// TIA Portal V16 export
// export: Created 2021-11-12T13:32:43.7602296Z, ExportSetting WithDefaults, DisplayName Totally Integrated Automation Portal, DisplayVersion V16 Update 3, DisplayName TIA Portal Version Control Interface, DisplayVersion V16 Update 2, DisplayName TIA Portal Openness, DisplayVersion V16 Update 3, DisplayName SINAMICS Startdrive Advanced, DisplayVersion V16 Update 5, DisplayName SINAMICS Startdrive G130, G150, S120, S150, SINAMICS MV, S210, DisplayVersion V16 Update 5, DisplayName SINAMICS Startdrive G110M, G120, G120C, G120D, G120P, G115D, DisplayVersion V16 Update 5, DisplayName STEP 7 Professional, DisplayVersion V16 Update 3, DisplayName STEP 7 Safety, DisplayVersion V16, DisplayName WinCC UA Professional, DisplayVersion V16 Update 3
DATA_BLOCK "STATUS_SCH1"   // DB51
{ S7_Optimized_Access := 'TRUE' }
VERSION : 0.1
// stored: AutoNumber true, DBAccessibleFromOPCUA true, IsOnlyStoredInLoadMemory false, IsRetainMemResEnabled false, IsWriteProtectedInAS false, MemoryReserve 100
   VAR
      xxxxx___BinarySensors___xxxxx : Byte;
      xxxxx___BinaryOthers___xxxxx : Byte;
      "000UH11-SF05_22" : Bool;   // Blokování lisu
      "000UH10-SF12_22" : Bool;   // Blokování lisu
      "TT1EB01-KF02_4" : Bool;   // Ohřev nástrojů 1 Kontrola chodu čerpadla
      "TT2EB01-KF02_4" : Bool;   // Ohřev nástrojů 2 Kontrola chodu čerpadla
      "200CM01-BL01_14" : Bool;   // Jímka pod lisem Plovák nahoře Varování
      "200CM01-BL01_12" : Bool;   // Jímka pod lisem Plovák dole OK
      xxxxx___AnalogueSensors___xxxxx : Byte;
      "TT1EB01-KF01_29" : Struct   // Tool heating 1 up actual temperature
         Main : "UDT_Status_main";
         Specific : "UDT_CH_AI_Status_specific";
         Error : "UDT_Error01";
      END_STRUCT;
      "TT1EB01-KF02_29" : Struct   // Tool heating 1 down actual temperature
         Main : "UDT_Status_main";
         Specific : "UDT_CH_AI_Status_specific";
         Error : "UDT_Error01";
      END_STRUCT;
      "TT2EB01-KF01_29" : Struct   // Tool heating 2 up actual temperature
         Main : "UDT_Status_main";
         Specific : "UDT_CH_AI_Status_specific";
         Error : "UDT_Error01";
      END_STRUCT;
      "TT2EB01-KF02_29" : Struct   // Tool heating 2 down actual temperature
         Main : "UDT_Status_main";
         Specific : "UDT_CH_AI_Status_specific";
         Error : "UDT_Error01";
      END_STRUCT;
      xxxxx___Drives___xxxxx : Byte;
      xxxxx___MaterialFlow___xxxxx : Byte;
   END_VAR
   VAR RETAIN
      MatCard : Array[1..7, 1..2] of "UDT_MatCard";   // Material card [Line - shorter side, Row - longer side]
   END_VAR
   VAR
      xxxxx___Other___xxxxx : Byte;
      "TT1EB01-KF01_27" : Struct   // Setpoint tool heating 1 up
         Main : "UDT_Status_main";
         Specific : "UDT_CH_AO_Status_specific";
         Error : "UDT_Error01";
      END_STRUCT;
      "TT1EB01-KF02_27" : Struct   // Setpoint tool heating 1 down
         Main : "UDT_Status_main";
         Specific : "UDT_CH_AO_Status_specific";
         Error : "UDT_Error01";
      END_STRUCT;
      "TT2EB01-KF01_27" : Struct   // Setpoint tool heating 2 up
         Main : "UDT_Status_main";
         Specific : "UDT_CH_AO_Status_specific";
         Error : "UDT_Error01";
      END_STRUCT;
      "TT2EB01-KF02_27" : Struct   // Setpoint tool heating 2 down
         Main : "UDT_Status_main";
         Specific : "UDT_CH_AO_Status_specific";
         Error : "UDT_Error01";
      END_STRUCT;
      Press : Struct   // Status of press machine
         Specific : "UDT_SCH_Status_specific";
      END_STRUCT;
      ToolTemperatureOK : Bool;   // Temperature of all tools is OK
      BrakeTestTime : Time_Of_Day;   // Remaining time to brake test - Press [min]
      xxxxx__Alarms___xxxxx : Byte;
      PressFault : Struct   // From press / Sumární porucha lisu.
         Main : "UDT_Status_main";
         Specific : "UDT_DI_Mon_Status_specific";
         Error { S7_SetPoint := 'True'} : "UDT_Error01";
      END_STRUCT;
      LiveBit : Struct   // Communication / Komunikace
         Main : "UDT_Status_main";
         Specific : "UDT_DI_Mon_Status_specific";
         Error { S7_SetPoint := 'True'} : "UDT_Error01";
      END_STRUCT;
      BrakeTestReqWrn : Struct   // Brake test required
         Main : "UDT_Status_main";
         Specific : "UDT_DI_Mon_Status_specific";
         Error { S7_SetPoint := 'True'} : "UDT_Error01";
      END_STRUCT;
      xxxxx___ProcessAlarms___xxxxx : Byte;
      "TT1EB01-KF01" : Struct   // Tool heating 1 up / Nahřívání nástrojů 1 nahoře.
         Main : "UDT_Status_main";
         Specific : "UDT_DI_Mon_Status_specific";
         Error { S7_SetPoint := 'True'} : "UDT_Error01";
      END_STRUCT;
      "TT1EB01-KF02" : Struct   // Tool heating 1 down / Nahřívání nástrojů 1 dole.
         Main : "UDT_Status_main";
         Specific : "UDT_DI_Mon_Status_specific";
         Error { S7_SetPoint := 'True'} : "UDT_Error01";
      END_STRUCT;
      "TT2EB01-KF01" : Struct   // Tool heating 2 up / Nahřívání nástrojů 2 nahoře.
         Main : "UDT_Status_main";
         Specific : "UDT_DI_Mon_Status_specific";
         Error { S7_SetPoint := 'True'} : "UDT_Error01";
      END_STRUCT;
      "TT2EB01-KF02" : Struct   // Tool heating 2 down / Nahřívání nástrojů 2 dole.
         Main : "UDT_Status_main";
         Specific : "UDT_DI_Mon_Status_specific";
         Error { S7_SetPoint := 'True'} : "UDT_Error01";
      END_STRUCT;
      "TT1EB01-KF02_3" : Struct   // Pump not running / Pumpa nejede.
         Main : "UDT_Status_main";
         Specific : "UDT_DI_Mon_Status_specific";
         Error { S7_SetPoint := 'True'} : "UDT_Error01";
      END_STRUCT;
      "TT2EB01-KF02_3" : Struct   // Pump not running / Pumpa nejede.
         Main : "UDT_Status_main";
         Specific : "UDT_DI_Mon_Status_specific";
         Error { S7_SetPoint := 'True'} : "UDT_Error01";
      END_STRUCT;
      "200CM01-BL01_15" : Struct   // Tank under press full / Jímka pod lisem Plovák nahoře Varování
         Main : "UDT_Status_main";
         Specific : "UDT_DI_Mon_Status_specific";
         Error { S7_SetPoint := 'True'} : "UDT_Error01";
      END_STRUCT;
      xxxxx__SafetyAlarms__xxxxx : Byte;
      ES : Struct   // E-stop SCH1
         Main : "UDT_Status_main";
         Specific { S7_SetPoint := 'True'} : "UDT_DI_Mon_Status_specific";
         Error { S7_SetPoint := 'True'} : "UDT_Error01";
      END_STRUCT;
   END_VAR
BEGIN
END_DATA_BLOCK
